// Mitsubishi GX Works2 project: git   PLC: Q02/Q02H

PROGRAM MAIN
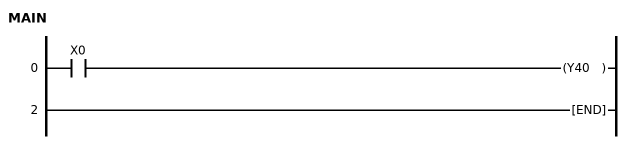
0     LD      X0
      OUT     Y40
2     END
END_PROGRAM
